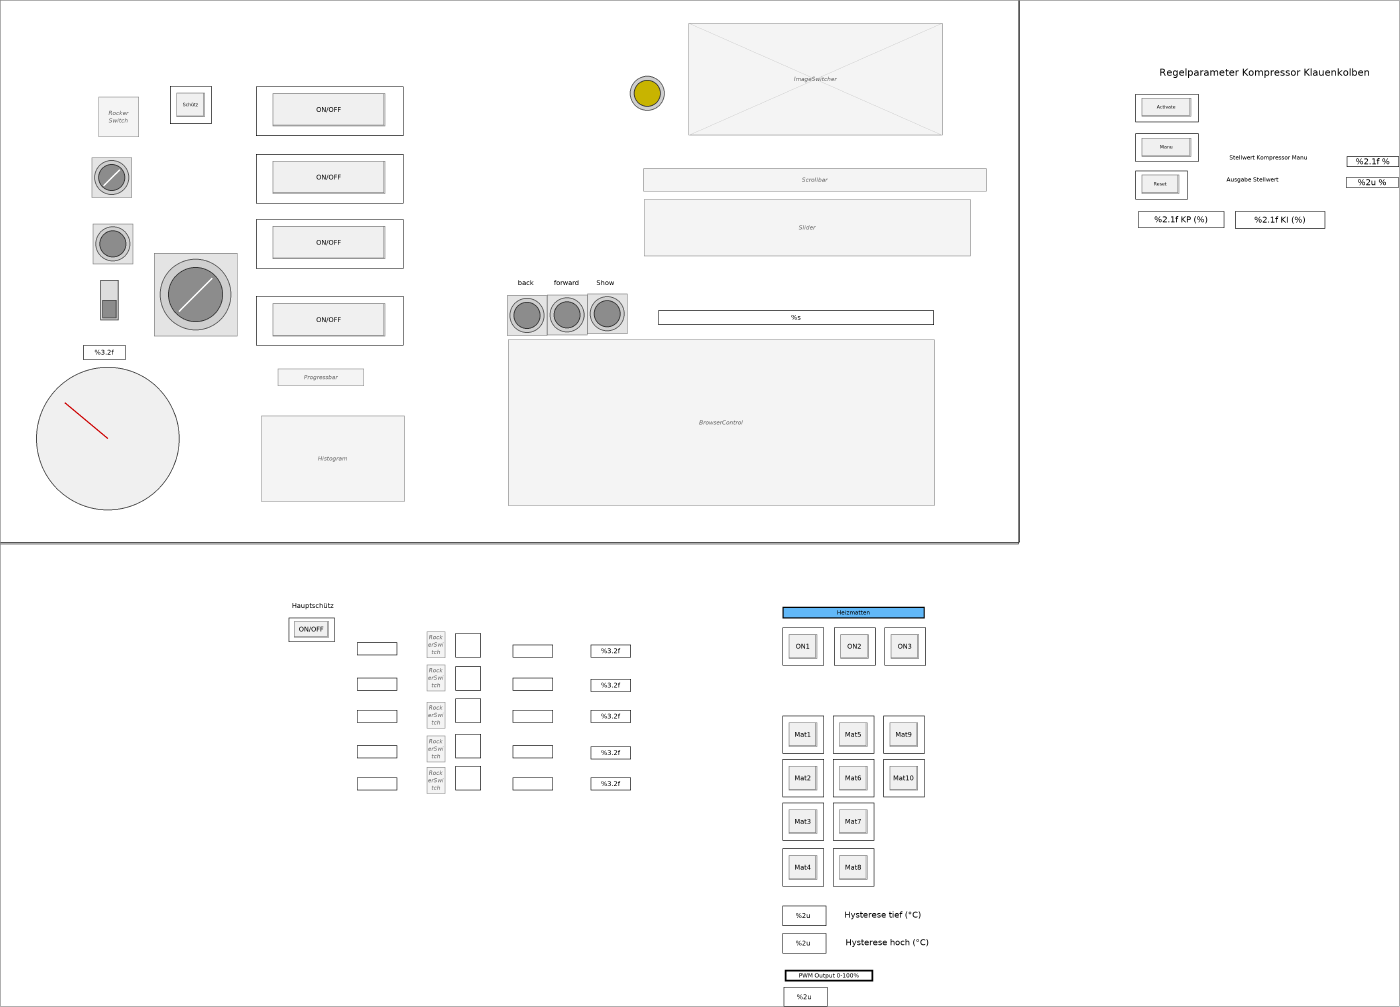
VISUALIZATION Testseite1  // 2444x1759, background image backround
    Rectangle (1778,0 2x947)
    Rectangle (0,947 1778x3)
    PushSwitchLed (162,391 70x70), variable: GVL.bManuHeat_REG3_CTRL, behaviour: TOGGLE, style: Switch-PushSwitchLed-Gray
    RockerSwitch (172,169 70x70), variable: GVL.bManuHeat_REG1_CTRL, behaviour: TOGGLE, style: Switch-RockerSwitch-Gray
    RotarySwitch (160,275 70x70), variable: GVL.bManuHeat_REG2_CTRL, behaviour: TOGGLE, style: Switch-RotarySwitch-Gray
    DipSwitch (156,489 70x70), variable: GVL.bManuHeat_REG4_CTRL, behaviour: TAP, style: Switch-DipSwitch-Gray
    Rectangle (447,269 257x86), colour toggle: GVL.bManuHeat_REG2_CTRL
    Button (476,281 196x57), "ON/OFF", pressed state: GVL.bManuHeat_REG2_CTRL
        toggle GVL.bManuHeat_REG2_CTRL
    Rectangle (447,151 257x86), colour toggle: GVL.bManuHeat_REG1_CTRL
    Button (476,163 196x57), "ON/OFF", pressed state: GVL.bManuHeat_REG1_CTRL
        toggle GVL.bManuHeat_REG1_CTRL
    Rectangle (447,383 257x86), colour toggle: GVL.bManuHeat_REG3_CTRL
    Button (476,395 196x57), "ON/OFF", pressed state: GVL.bManuHeat_REG3_CTRL
        toggle GVL.bManuHeat_REG3_CTRL
    Rectangle (447,517 257x86), colour toggle: GVL.bManuHeat_REG4_CTRL
    Button (476,530 196x57), "ON/OFF", pressed state: GVL.bManuHeat_REG4_CTRL
        toggle GVL.bManuHeat_REG4_CTRL
    Lamp1 (1095,128 70x70), style: Lamp-Lamp1-Yellow
    BrowserControl (887,593 744x290)
        p3734058945: SurlAdress
        p2179181546: bShow
        p2928617338: bBack
        p728663958: bForward
    PushSwitchLed (885,516 70x70), variable: bForward, behaviour: TAP, style: Switch-PushSwitchLed-Gray
    PushSwitchLed (955,515 70x70), variable: bBack, behaviour: TAP, style: Switch-PushSwitchLed-Gray
    PushSwitchLed (1025,513 70x70), variable: bShow, behaviour: TAP, style: Switch-PushSwitchLed-Gray
    Rectangle (886,479 64x30), "back"
    Rectangle (957,479 64x30), "forward"
    Rectangle (1025,479 64x30), "Show"
    Rectangle (1149,542 481x25), "%s", tooltip "Durchmesser in mm eingeben", text variable: SurlAdress
        OnMouseDown: write the text variable via Edit, min 0, max 150
    Histogram (456,726 250x150), scale format: %.1f, scale 0..100
        p1518820177: aArray_Histogram
        p102497268: aArray_Histogram
        p788070771: ARRAY [0..100] OF INT
    Meter360 (63,641 250x250), value: Istwert_IN_NV_OUT, style: Meter-Meter360-Gray, scale format: %.1f, scale 0..100
    Rectangle (145,603 74x25), "%3.2f", tooltip "Durchmesser in mm eingeben", text variable: GVL.fSetpointValue1
        OnMouseDown: write the text variable via VisuDialogs.Numpad, min 0, max 150
    Slider (1124,348 570x99), variable: GVL.fSetpointValue1, scale 0..100
    Scrollbar (1123,294 599x40)
        p1057716461: GVL.fSetpointValue1
    Progressbar (485,644 150x30)
    Potentiometer360 (269,429 145x171), variable: GVL.fSetpointValue1, style: Potentiometer-Potentiometer360-Gray, scale format: %.1f, scale 0..100
        p2431819421: Outside
    Group (623,1103 478x283)
        Rectangle (0,81 70x22), colour toggle: GVL.bAuto_Heat_REG5_CTRL
        Rectangle (272,81 70x22), colour toggle: GVL.HEAT_Reg_5_OUT
        Rectangle (0,19 70x22), colour toggle: GVL.bAuto_Heat_REG4_CTRL
        Rectangle (272,23 70x22), colour toggle: GVL.HEAT_Reg_4_OUT
        Rectangle (408,83 70x22), "%3.2f", text variable: GVL.fPWMDutyCycle5
        Rectangle (408,23 70x22), "%3.2f", text variable: GVL.fPWMDutyCycle4
        Rectangle (0,137 70x22), colour toggle: GVL.bAuto_Heat_REG6_CTRL
        Rectangle (272,137 70x22), colour toggle: GVL.HEAT_Reg_6_OUT
        Rectangle (408,137 70x22), "%3.2f", text variable: GVL.fPWMDutyCycle6
        Rectangle (0,199 70x22), colour toggle: GVL.bAuto_Heat_REG7_CTRL
        Rectangle (272,199 70x22), colour toggle: GVL.HEAT_Reg_7_OUT
        Rectangle (408,201 70x22), "%3.2f", text variable: GVL.fPWMDutyCycle7
        Rectangle (0,255 70x22), colour toggle: GVL.bAuto_Heat_REG8_CTRL
        Rectangle (172,61 44x42), colour toggle: GVL.bManuHeat_REG5_CTRL
        Rectangle (172,3 44x42), colour toggle: GVL.bManuHeat_REG4_CTRL
        Rectangle (172,117 44x42), colour toggle: GVL.bManuHeat_REG6_CTRL
        Rectangle (172,179 44x42), colour toggle: GVL.bManuHeat_REG7_CTRL
        Rectangle (172,235 44x42), colour toggle: GVL.bManuHeat_REG8_CTRL
        Rectangle (272,255 70x22), colour toggle: GVL.HEAT_Reg_8_OUT
        Rectangle (408,255 70x22), "%3.2f", text variable: GVL.fPWMDutyCycle8
        RockerSwitch (122,0 32x46), variable: GVL.bManuHeat_REG4_CTRL, behaviour: TOGGLE, style: Switch-RockerSwitch-Gray
        RockerSwitch (122,58 32x46), variable: GVL.bManuHeat_REG5_CTRL, behaviour: TOGGLE, style: Switch-RockerSwitch-Gray
        RockerSwitch (122,123 32x46), variable: GVL.bManuHeat_REG6_CTRL, behaviour: TOGGLE, style: Switch-RockerSwitch-Gray
        RockerSwitch (122,182 32x46), variable: GVL.bManuHeat_REG7_CTRL, behaviour: TOGGLE, style: Switch-RockerSwitch-Gray
        RockerSwitch (122,237 32x46), variable: GVL.bManuHeat_REG8_CTRL, behaviour: TOGGLE, style: Switch-RockerSwitch-Gray
    Rectangle (504,1079 80x42), colour toggle: GVL.HEAT_Reg_Mainswitch_OUT
    Button (513,1085 61x28), "ON/OFF", pressed state: GVL.HEAT_Reg_Mainswitch_Manu
        toggle GVL.HEAT_Reg_Mainswitch_Manu
    Rectangle (500,1043 92x30), "Hauptschütz"
    Group (1366,1060 270x699)
        Rectangle (0,190 72x66), colour toggle: GVL.Heat_matt1
        Button (11,202 49x42), "Mat1", pressed state: GVL.Heat_matt1_manu
            toggle GVL.Heat_matt1_manu
        Rectangle (88,266 72x66), colour toggle: GVL.Heat_matt6
        Button (99,278 49x42), "Mat6", pressed state: GVL.Heat_matt6_manu
            toggle GVL.Heat_matt6_manu
        Rectangle (0,266 72x66), colour toggle: GVL.Heat_matt2
        Button (11,278 49x42), "Mat2", pressed state: GVL.Heat_matt2_manu
            toggle GVL.Heat_matt2_manu
        Rectangle (88,342 72x66), colour toggle: GVL.Heat_matt7
        Button (99,354 49x42), "Mat7", pressed state: GVL.Heat_matt7_manu
            toggle GVL.Heat_matt7_manu
        Rectangle (0,342 72x66), colour toggle: GVL.Heat_matt3
        Button (11,354 49x42), "Mat3", pressed state: GVL.Heat_matt3_manu
            toggle GVL.Heat_matt3_manu
        Rectangle (88,422 72x66), colour toggle: GVL.Heat_matt8
        Button (99,434 49x42), "Mat8", pressed state: GVL.Heat_matt8_manu
            toggle GVL.Heat_matt8_manu
        Rectangle (0,422 72x66), colour toggle: GVL.Heat_matt4
        Button (11,434 49x42), "Mat4", pressed state: GVL.Heat_matt4_manu
            toggle GVL.Heat_matt4_manu
        Rectangle (176,190 72x66), colour toggle: GVL.Heat_matt9
        Button (187,202 49x42), "Mat9", pressed state: GVL.Heat_matt9_manu
            toggle GVL.Heat_matt9_manu
        Rectangle (88,190 72x66), colour toggle: GVL.Heat_matt5
        Button (99,202 49x42), "Mat5", pressed state: GVL.Heat_matt5_manu
            toggle GVL.Heat_matt5_manu
        Rectangle (176,266 72x66), colour toggle: GVL.Heat_matt10
        Button (187,278 49x42), "Mat10", pressed state: GVL.Heat_matt10_manu
            toggle GVL.Heat_matt10_manu
        Rectangle (0,0 248x20), "Heizmatten"
        Rectangle (178,36 72x66), colour toggle: GVL.Switch_Heat_group3
        Button (189,48 49x42), "ON3", pressed state: GVL.Switch_Heat_group3
            toggle GVL.Switch_Heat_group3
        Rectangle (90,36 72x66), colour toggle: GVL.Switch_Heat_group2
        Button (101,48 49x42), "ON2", pressed state: GVL.Switch_Heat_group2
            toggle GVL.Switch_Heat_group2
        Rectangle (0,36 72x66), colour toggle: GVL.Switch_Heat_group1
        Button (11,48 49x42), "ON1", pressed state: GVL.Switch_Heat_group1
            toggle GVL.Switch_Heat_group1
        Rectangle (2,664 76x35), "%2u", tooltip "Durchmesser in mm eingeben", text variable: GVL.PWM_duty_cycle
            OnMouseDown: write the text variable via VisuDialogs.Numpad, min 0, max 100
        Rectangle (4,634 154x20), "PWM Output 0-100%"
        Rectangle (0,522 76x35), "%2u", tooltip "Durchmesser in mm eingeben", text variable: GVL.Hyst_low_LIM_Heatmatt
            OnMouseDown: write the text variable via VisuDialogs.Numpad, min 0, max 150
        Rectangle (0,570 76x35), "%2u", tooltip "Durchmesser in mm eingeben", text variable: GVL.Hyst_high_LIM_Heatmatt
            OnMouseDown: write the text variable via VisuDialogs.Numpad, min 0, max 150
        Rectangle (94,522 162x32), "Hysterese tief (°C)"
        Rectangle (96,570 174x32), "Hysterese hoch (°C)"
    Rectangle (297,150 72x66), colour toggle: GVL.M_Belt_Feeder_Switch_ON_Manu
    Button (308,162 49x42), "Schütz", pressed state: GVL.M_Belt_Feeder_Switch_ON_Manu
        toggle GVL.M_Belt_Feeder_Switch_ON_Manu
    Rectangle (1972,110 472x33), "Regelparameter Kompressor Klauenkolben"
    Rectangle (2351,273 91x18), "%2.1f %", tooltip "Durchmesser in mm eingeben", text variable: GVL.fManual_controller_Primaer_comp
        OnMouseDown: write the text variable via VisuDialogs.Numpad, min 0, max 100
    Rectangle (1982,233 110x49), colour toggle: GVL.Set_Manual_controller_Primaer_comp
    Button (1993,241 86x32), "Manu", pressed state: GVL.Set_Manual_controller_Primaer_comp
        toggle GVL.Set_Manual_controller_Primaer_comp
    Rectangle (2350,309 91x19), "%2u %", tooltip "Durchmesser in mm eingeben", text variable: GVL.fStellwert_Primaer_comp
    Rectangle (2097,305 179x17), "Ausgabe Stellwert"
    Rectangle (1982,298 91x50), colour toggle: GVL.Reset_Controller_Primaer_comp
    Button (1993,305 65x33), "Reset"
        tap GVL.Reset_Controller_Primaer_comp
    Rectangle (1987,369 150x29), "%2.1f KP (%)", tooltip "Durchmesser in mm eingeben", text variable: GVL.fKP_Controller_Primaer_comp
        OnMouseDown: write the text variable via VisuDialogs.Numpad, min 0, max 100
    Rectangle (2156,369 157x30), "%2.1f KI (%)", tooltip "Durchmesser in mm eingeben", text variable: GVL.fKI_Controller_Primaer_comp
        OnMouseDown: write the text variable via VisuDialogs.Numpad, min 0, max 100
    Rectangle (2103,266 223x18), "Stellwert Kompressor Manu"
    Rectangle (1982,164 110x49), colour toggle: GVL.Activate_controller_Primaer_comp
    Button (1993,171 86x32), "Activate", pressed state: GVL.Activate_controller_Primaer_comp
        toggle GVL.Activate_controller_Primaer_comp
    ImageSwitcher (1202,40 443x196), background image: Triss_PID_V5, image: AQ, behaviour: TOGGLE
        p3148411668: LAyout
END_VISUALIZATION

(* stored: Version 1.1.0.1, ProductVersion 3.1.4024.3
   Visu Testseite1: Id {3019dc83-d84d-4afe-86a3-965b0a29327a} *)
